// TwinCAT 3 PLC project PLC
// ProgramVersion: 3.1.4026.21
// libraries:
//   Tc2_MC2, * (Beckhoff Automation GmbH)
//   Tc2_Standard, * (Beckhoff Automation GmbH)
//   Tc2_System, * (Beckhoff Automation GmbH)
//   Tc3_IotBase, * (Beckhoff Automation GmbH)
// project tree:
//   DUTs/ E_State.TcDUT
//   GVLs/ IFC_HW.TcGVL
//   / PlcTask.TcTTO
//   POUs/ FB_Abfuellmodul.TcPOU, FB_CNV.TcPOU, FB_Dispenser.TcPOU, FB_IOT.TcPOU, FB_Man_X.TcPOU, FB_RCrtl.TcPOU, FB_StatusLight.TcPOU, FB_TimeOutError.TcPOU, FB_Transport.TcPOU, FB_Vereinzelung.TcPOU, MAIN.TcPOU
// (motion and I/O tree: see PLC project tempmodel)
// real-time tasks:
//   TASK PlcTask: cycle T#10ms, priority 21, ADS port 350
//   TASK PlcTask1: cycle T#10ms, priority 22, ADS port 351
//   TASK PlcTask2: cycle T#10ms, priority 20, ADS port 352
// variable links:
//   LF_System_PLC/LF_System_PLC Instance <-> PLC/PLC Instance
//     PlcTask Inputs/MAIN.bIN_Gripper <-> PlcTask Outputs/IFC_HW.bGripperClosed
//     PlcTask Inputs/MAIN.bIN_Stopper1 <-> PlcTask Outputs/IFC_HW.bBandHub1
//     PlcTask Inputs/MAIN.bIN_Stopper2 <-> PlcTask Outputs/IFC_HW.bBandHub2
//     PlcTask Inputs/MAIN.bIN_Stopper3 <-> PlcTask Outputs/IFC_HW.bBandHub3
//     PlcTask Inputs/MAIN.bIn_LedGreen <-> PlcTask Outputs/IFC_HW.bAmpelGrun
//     PlcTask Inputs/MAIN.bIn_LedRot <-> PlcTask Outputs/IFC_HW.bAmpelRot
//     PlcTask Inputs/MAIN.bIn_LedYellow <-> PlcTask Outputs/IFC_HW.bAmpelGelb
//     PlcTask Inputs/MAIN.bIn_Schleuse1_L1 <-> PlcTask Outputs/IFC_HW.bR1AKT1
//     PlcTask Inputs/MAIN.bIn_Schleuse1_L2 <-> PlcTask Outputs/IFC_HW.bR2AKT1
//     PlcTask Inputs/MAIN.bIn_Schleuse2_L1 <-> PlcTask Outputs/IFC_HW.bR1AKT2
//     PlcTask Inputs/MAIN.bIn_Schleuse2_L2 <-> PlcTask Outputs/IFC_HW.bR2AKT2
//     PlcTask Outputs/MAIN.bEnable <-> PlcTask Inputs/IFC_HW.bEnable
//     PlcTask Outputs/MAIN.bExecute <-> PlcTask Inputs/IFC_HW.bExecute
//     PlcTask Outputs/MAIN.bOUT_CnvNS{1..4} <-> PlcTask Inputs/IFC_HW.bBandSens{1..4}  (4 links)
//     PlcTask Outputs/MAIN.bOUT_SensMaxX <-> PlcTask Inputs/IFC_HW.bManEndXmax
//     PlcTask Outputs/MAIN.bOUT_SensMinX <-> PlcTask Inputs/IFC_HW.bManEndXmin
//     PlcTask Outputs/MAIN.bOut_VereinzelungNS1 <-> PlcTask Inputs/IFC_HW.bEinzelSens1
//     PlcTask Outputs/MAIN.bOut_VereinzelungNS2 <-> PlcTask Inputs/IFC_HW.bEinzelSens2
//     PlcTask Outputs/MAIN.bOut_VereinzelungNS3 <-> PlcTask Inputs/IFC_HW.bEinzelSens3
//     PlcTask Outputs/MAIN.iOut_USS1 <-> PlcTask Inputs/IFC_HW.iFillSens1
//     PlcTask Outputs/MAIN.iOut_USS2 <-> PlcTask Inputs/IFC_HW.iFillSens2
//     PlcTask Outputs/MAIN.iOut_USS3 <-> PlcTask Inputs/IFC_HW.iFillSens3
//   PLC/PLC Instance <-> NC-Task 1 SAF/Axes/BandAchse
//     PlcTask Inputs/IFC_HW.ax_BandMotor.NcToPlc <-> Outputs/ToPlc
//     PlcTask Outputs/IFC_HW.ax_BandMotor.PlcToNc <-> Inputs/FromPlc
//   PLC/PLC Instance <-> NC-Task 1 SAF/Axes/Extruder1
//     PlcTask Inputs/IFC_HW.ax_Extruder1.NcToPlc <-> Outputs/ToPlc
//     PlcTask Outputs/IFC_HW.ax_Extruder1.PlcToNc <-> Inputs/FromPlc
//   PLC/PLC Instance <-> NC-Task 1 SAF/Axes/Extruder2
//     PlcTask Inputs/IFC_HW.ax_Extruder2.NcToPlc <-> Outputs/ToPlc
//     PlcTask Outputs/IFC_HW.ax_Extruder2.PlcToNc <-> Inputs/FromPlc
//   PLC/PLC Instance <-> NC-Task 1 SAF/Axes/Extruder3
//     PlcTask Inputs/IFC_HW.ax_Extruder3.NcToPlc <-> Outputs/ToPlc
//     PlcTask Outputs/IFC_HW.ax_Extruder3.PlcToNc <-> Inputs/FromPlc
//   PLC/PLC Instance <-> NC-Task 1 SAF/Axes/X_Achse_Manipulator
//     PlcTask Inputs/IFC_HW.ax_ManX.NcToPlc <-> Outputs/ToPlc
//     PlcTask Outputs/IFC_HW.ax_ManX.PlcToNc <-> Inputs/FromPlc

CONFIGURATION PLC
    RESOURCE PLC ON TwinCAT3
        TASK PlcTask(INTERVAL := T#10ms, PRIORITY := 20);
        PROGRAM MAIN WITH PlcTask : MAIN;
    END_RESOURCE
END_CONFIGURATION

// ---- DUTs/E_State.TcDUT
{attribute 'qualified_only'}
{attribute 'strict'}
{attribute 'to_string'}
TYPE E_State :
(
    Off,
    Init,
    Ready,
    Production,
    Done,
    Error,
    Stop,
    Setup
);
END_TYPE

// ---- GVLs/IFC_HW.TcGVL
// In dieser GVL werden alle Variablen deklariert die auf die realen Klemmen zugreifen
VAR_GLOBAL
	
	// Allgemeine Variablen fur MAIN und HMI
		bEnable		AT%I*	: BOOL;			// Enable Factory (HMI Production Umgebung)
		bExecute	AT%I*	: BOOL;			// Startsignal	(Start Knopf Konsole)
		bStop				: BOOL;			// Stop Variable (interne Variable um FB's zu stoppen)
		bReset 				: bool; 		// Reset neu hinzugefgt
		
	// Station Statusampel	
		bAmpelRot 	AT%Q* 	: BOOL;			// Signal-LED Rot
		bAmpelGelb 	AT%Q* 	: BOOL;			// Signal-LED Gelb
		bAmpelGrun 	AT%Q* 	: BOOL;			// Signal-LED Grun
			
	// Station Vereinzelung
		bEinzelSens1 	AT%I*	: BOOL;					// Separation Sensor 1 (Kammer)
		bEinzelSens2 	AT%I*	: BOOL;					// Separation Sensor 2 (Rohr)
		bEinzelSens3 	AT%I*	: BOOL;					// Separation Sensor 3 (Flasche auf Kopf)
		bR1AKT1 		AT%Q* 	: BOOL := FALSE;		// Relais 1 Aktor 1 (Schleuse Oben öffnen)
		bR2AKT1 		AT%Q* 	: BOOL := TRUE; 		// Relais 2 Aktor 1 (Schleuse Oben schließen)
		bR1AKT2 		AT%Q* 	: BOOL := FALSE;		// Relais 1 Aktor 2 (Schleuse Unten öffne)
		bR2AKT2 		AT%Q* 	: BOOL := TRUE;			// Relais 2 Aktor 2	(Schleuse Unten schließen)
	
	// Station Forderband
		bBandSens1 	AT %I*	: BOOL;		// Forderband Sensor 1 (Extruder 1)
		bBandSens2	AT %I*	: BOOL;		// Forderband Sensor 2 (Extruder 2)
		bBandSens3 	AT %I*	: BOOL;		// Forderband Sensor 3 (Extruder 3)
		bBandSens4 	AT %I*	: BOOL;		// Forderband Sensor 4 (Übergabe Roboter)
		bBandHub1 	AT %Q*	: BOOL;		// Forderband Hubmagnet 1 (Schleuse Extruder 1)
		bBandHub2 	AT %Q*	: BOOL;		// Forderband Hubmagnet 1 (Schleuse Extruder 2)
		bBandHub3 	AT %Q*	: BOOL;		// Forderband Hubmagnet 1 (Schleuse Extruder 3)
		
		ax_Extruder1 	: AXIS_REF;		// Forderband NC-Achse Extruder 1
		ax_Extruder2 	: AXIS_REF;		// Forderband NC-Achse Extruder 2
		ax_Extruder3 	: AXIS_REF;		// Forderband NC-Achse Extruder 3
		ax_BandMotor 	: AXIS_REF;		// Forderband NC-Achse Band
		
		iBandFullmenge1		: INT := 1;	// in Gramm (Soll Füllmenge Extruder 1)
		iBandFullmenge2		: INT := 1;	// in Gramm (Soll Füllmenge Extruder 2)
		iBandFullmenge3		: INT := 1;	// in Gramm (Soll Füllmenge Extruder 3)
		
	//Füllstandsüberwachung
		iFillSens1 AT%I*	: UINT;		// Füllstandssensor im Granulatspeicher 1
		iFillSens2 AT%I*	: UINT;		// Füllstandssensor im Granulatspeicher 2
		iFillSens3 AT%I*	: UINT;		// Füllstandssensor im Granulatspeicher 3
		
		rFillLevelPercent1	: REAL;		// Füllstand im Granulatspeicher 1 in %
		rFillLevelGramm1	: REAL;		// Füllstand im Granulatspeicher 1 in g
		rFillLevelPercent2	: REAL;		// Füllstand im Granulatspeicher 2 in %
		rFillLevelGramm2	: REAL;		// Füllstand im Granulatspeicher 2 in g
		rFillLevelPercent3	: REAL;		// Füllstand im Granulatspeicher 3 in %
		rFillLevelGramm3	: REAL;		// Füllstand im Granulatspeicher 3 in g
		
		rMaxFillLevel 		: REAL := 375;	// Kalibrierter Füllstand für 10% * 10
		
	// Station Waage
		sWaageNachricht		: STRING;	// Nachricht von Wagezelle (fur virtuelle Inbetriebnahme notig)
		bWaageNull			: BOOL;		// TARA Waage (Waage auf Null setzen)
		iWaageMesswert		: INT;		// Messwert der Waage
		
	// Station Behalteridentifikation
		bIdSensorTrager		: BOOL;		// Sensor bei Erkennung eines Datentrager
		sIdNachricht		: STRING;	// Nachricht von RFID-System (fur virtuelle Inbetriebnahme notig)
		sSeriennummer		: STRING;	// Seriennummer RFID-Tag
		
	//Temperierstation
		bVentilator1 	AT %Q*	: BOOL;		// Ventilator 1
		bVentilator2 	AT %Q*	: BOOL;		// Ventilator 2
		bVentilator3 	AT %Q*	: BOOL;		// Ventilator 3
		
		iTempSens1 		AT%I*	: UINT;		// Temperatursensor 1
		iTempSens2 		AT%I*	: UINT;		// Temperatursensor 2
		iHeizpatrone 	AT%Q*	: UINT;		// Heizpatronen
		
		iMaxTemp				: UINT := 5500;		// in °C * 100
		
	// Station Manipulator
		bManEndXmin 		AT%I* 	: BOOL := TRUE;		// Manipulator min Endschalter Achse x
		bManEndYmin 		AT%I* 	: BOOL := TRUE;		// Manipulator min Endschalter Achse y
		bManEndZmin 		AT%I* 	: BOOL := TRUE;		// Manipulator min Endschalter Achse z
		bManEndGmin 		AT%I* 	: BOOL := TRUE;		// Manipulator min Endschalter Achse Gripper
		bManEndXmax 		AT%I* 	: BOOL := TRUE;		// Manipulator max Endschalter Achse x
		bManEndYmax 		AT%I* 	: BOOL := TRUE;		// Manipulator max Endschalter Achse y
		bManEndZmax 		AT%I* 	: BOOL := TRUE;		// Manipulator max Endschalter Achse z
		bManEndGmax 		AT%I* 	: BOOL := TRUE;		// Manipulator max Endschalter Achse Gripper
		bManBrakeZ			AT%Q*	: BOOL := FALSE;	// Bremse Achse z
		
		ax_ManX			: AXIS_REF;			// Manipulator NC-Achse x
		ax_ManY			: AXIS_REF;			// Manipulator NC-Achse y
		ax_ManZ			: AXIS_REF;			// Manipulator NC-Achse z
		ax_ManG			: AXIS_REF; 		// Manipulator NC-Achse Gripper
		
		bGripperClosed		AT%Q*	: BOOL; 			// signal if gripper is closed ONLY USED IN SIM
END_VAR

// ---- POUs/MAIN.TcPOU
PROGRAM MAIN
VAR
	// Die Logik-Bausteine (Module Level)
    fbAmpel        : FB_StatusLight;
    //fbVereinzelung : FB_Vereinzelung;
    //fbTransport    : FB_Transport;
    
    // NEU: Die drei Abfüllstationen (Dispenser)
    //fbDisp1        : FB_Dispenser;
    //fbDisp2        : FB_Dispenser;
    //fbDisp3        : FB_Dispenser;

    // NEU: Der Werksleiter / Master (Machine Level)
    // Er steuert die oben genannten Module
    fbModul        : FB_Abfuellmodul;
	fbManX         : FB_Man_X;
    // Die Hardware-Übersetzer für die Relais (Process Level)
//     fbRelaisZyl1   : FB_RCrtl; // Schleuse oben
//     fbRelaisZyl2   : FB_RCrtl; // Schleuse unten
    
    // Der Antrieb
    //fbBand         : FB_CNV;
	fbiot : FB_IOT;
	
	//reset
	reset : BOOL;
	bError : Bool;
END_VAR

// --- 1. DER CHEF GIBT DIE BEFEHLE (Hierarchisches Modul) ---

fbiot(iUSS1 := IFC_HW.iFillSens1, iUSS2 := IFC_HW.iFillSens2, iUSS3 := IFC_HW.iFillSens3);
//fbiot(iUSS1 := iIn_USS1, iUSS2 := iIn_USS2, iUSS3 := iIn_USS3);


fbModul(
    bEnable := IFC_HW.bEnable,
    bExecute := IFC_HW.bExecute,
	//bTransportError := fbTransport.bError, 
    bReset := reset,
    
    // Status-Rückmeldungen der Arbeiter abfragen
    //bVereinzelungDone := (fbVereinzelung.eStateOut = E_State.Done),
    //bTransportDone    := (fbTransport.eState = E_State.Done),
    //bDisp1Done        := (fbDisp1.eState = E_State.Done),
    //bDisp2Done        := (fbDisp2.eState = E_State.Done),
    //bDisp3Done        := (fbDisp3.eState = E_State.Done)
);


fbManX(
    // Steuerbefehle
    bEnable         := ifc_hw.bEnable,
    bExecute        := ifc_hw.bExecute, // Hier ggf. eine andere Variable nehmen, wenn er unabhängig vom Abfüllmodul starten soll!
    bHalt           := FALSE,           // Aktuell nicht extern genutzt, ggf. anpassen
    
    // Hardware-Sensoren (Endschalter)
    bEndSchalterMin := ifc_hw.bManEndXmin, 
    bEndSchalterMax := ifc_hw.bManEndXmax, // Falls vorhanden, sonst FALSE
    
    // Fahrparameter (Können später auch aus einer Rezeptur/HMI kommen)
    fPosition       := -500.0,  // Zielposition (Beispiel)
    fVelocity       := 30.0,  // Zielgeschwindigkeit
    pHome           := 0.0,   // Referenzposition am linken Anschlag
    
    // Verknüpfung zur NC-Achse
    ax              := ifc_hw.ax_ManX
);

// --- 2. DIE ARBEITER FÜHREN AUS ---

// Vereinzelung
// fbVereinzelung(
//     bEnable  := IFC_HW.bEnable,
//     bExecute := fbModul.bStartVereinzelung,
//     bSens1   := IFC_HW.bEinzelSens1,
//     bSens2   := IFC_HW.bEinzelSens2,
//     bSens3   := IFC_HW.bEinzelSens3
// );

// Ampel und Relais für Vereinzelung
fbAmpel(eState := fbModul.eState);
IFC_HW.bAmpelRot   := fbAmpel.bLightRed;
IFC_HW.bAmpelGelb  := fbAmpel.bLightYellow;
IFC_HW.bAmpelGrun  := fbAmpel.bLightGreen;

// fbRelaisZyl1(bIn := fbModul.fbVereinzelung.bGate1);
// fbRelaisZyl2(bIn := fbModul.fbVereinzelung.bGate2);
// IFC_HW.bR1AKT1 := fbRelaisZyl1.bQ1;
// IFC_HW.bR2AKT1 := fbRelaisZyl1.bQ2;
// IFC_HW.bR1AKT2 := fbRelaisZyl2.bQ1;
// IFC_HW.bR2AKT2 := fbRelaisZyl2.bQ2;

// Transport-Management
// fbTransport(
//     bEnable  := IFC_HW.bEnable,
//     bExecute := fbModul.bStartTransport,    // <-- Befehl kommt vom Chef
// 	bReset   := reset,
//     nStation := fbModul.nZielStation,       // <-- Ziel (1, 2, 3, 4) kommt vom Chef
//     bSens1   := IFC_HW.bBandSens1,
//     bSens2   := IFC_HW.bBandSens2,
//     bSens3   := IFC_HW.bBandSens3,
//     bSens4   := IFC_HW.bBandSens4
// );

// Die Band-Stopper
// IFC_HW.bBandHub1 := fbTransport.bHub1;
// IFC_HW.bBandHub2 := fbTransport.bHub2;
// IFC_HW.bBandHub3 := fbTransport.bHub3;


// --- 3. DIE EXTRUDER ---

// fbDisp1(
//     ax := IFC_HW.ax_Extruder1,
//     bEnable := IFC_HW.bEnable,
//     bExecute := fbModul.bStartDisp1,        // <-- Befehl kommt vom Chef
//     bSensFlasche := IFC_HW.bBandSens1,
//     iFuellstand := IFC_HW.iFillSens1,
//     iLimit := 80                            // Hier könntest du später Variablen einsetzen
// );
// 
// fbDisp2(
//     ax := IFC_HW.ax_Extruder2,
//     bEnable := IFC_HW.bEnable,
//     bExecute := fbModul.bStartDisp2,        // <-- Befehl kommt vom Chef
//     bSensFlasche := IFC_HW.bBandSens2,
//     iFuellstand := IFC_HW.iFillSens2,
//     iLimit := 80
// );
// 
// fbDisp3(
//     ax := IFC_HW.ax_Extruder3,
//     bEnable := IFC_HW.bEnable,
//     bExecute := fbModul.bStartDisp3,        // <-- Befehl kommt vom Chef
//     bSensFlasche := IFC_HW.bBandSens3,
//     iFuellstand := IFC_HW.iFillSens3,
//     iLimit := 80
// );


// --- 4. DER MUSKEL FÜRS BAND ---

// fbBand(
//     bEnable  := IFC_HW.bEnable,        
//     bExecute := fbModul.fbTransport.bBandExecute, // Fahrbefehl vom Transport-Baustein
//     bHalt    := fbModul.fbTransport.bBandHalt,    // Bremsbefehl vom Transport-Baustein
//     rVel     := 50.0,                 
//     ax       := IFC_HW.ax_BandMotor    
// );

bError := (fbModul.eState = E_State.Error); 	// Überprüfen ob Fehler
ifc_hw.breset := reset;
IF reset AND NOT bError THEN 
	ifc_hw.bStop := FALSE;
	reset := FALSE;
END_IF

END_PROGRAM

// ---- POUs/FB_StatusLight.TcPOU
FUNCTION_BLOCK FB_StatusLight
VAR_INPUT
    eState : E_State;
END_VAR
VAR_OUTPUT
	bLightRed    : BOOL;
    bLightYellow : BOOL;
    bLightGreen  : BOOL;
END_VAR
VAR
	fbTimer      : TON;   // Timer
    bBlinkSignal : BOOL;  // Wechsel
END_VAR

// Grundstellung -> alles aus
bLightRed    := FALSE;
bLightYellow := FALSE;
bLightGreen  := FALSE;

// Blink Signal
fbTimer(IN := NOT fbTimer.Q, PT := T#500MS);
IF fbTimer.Q THEN
    bBlinkSignal := NOT bBlinkSignal;
END_IF

// Blink Zustände
CASE eState OF
    E_State.Off:
        bLightRed := TRUE;
        
    E_State.Production:
        bLightGreen := TRUE;
        
    E_State.Done:
        bLightYellow := TRUE;
        bLightGreen  := TRUE;
	
	E_State.Error:
        bLightRed := bBlinkSignal; // Rot blinken
        
    E_State.Stop:
        bLightRed    := bBlinkSignal; // Rot und Gelb blinken
        bLightYellow := bBlinkSignal;
        
    E_State.Init:
        bLightGreen := bBlinkSignal; // Grün blinken
        
    E_State.Ready:
        bLightYellow := bBlinkSignal; // Gelb und Grün blinken
        bLightGreen  := bBlinkSignal;
        
    E_State.Setup:
        bLightYellow := bBlinkSignal; // Gelb blinken
END_CASE

END_FUNCTION_BLOCK

// ---- POUs/FB_Abfuellmodul.TcPOU
FUNCTION_BLOCK FB_Abfuellmodul
VAR_INPUT
    bEnable  : BOOL;
    bExecute : BOOL;
    bReset   : BOOL;
    
    // Status-Rückmeldungen der Abteilungsleiter
    // bVereinzelungDone : BOOL;
    // bTransportDone    : BOOL;
    // bDisp1Done        : BOOL;
    // bDisp2Done        : BOOL;
    // bDisp3Done        : BOOL;
    
    // Error handling
    //bTransportError : BOOL; 
END_VAR
VAR_OUTPUT
    eState   : E_State;
END_VAR
VAR
    nState : INT;
    i      : INT; // Unser Stations-Zähler (1, 2, 3)
    bFlascheAktiv : BOOL;    // Flasche im System?
    
    fbVereinzelung : FB_Vereinzelung; 
    fbTransport    : FB_Transport;
    fbDisp1        : FB_Dispenser;
    fbDisp2        : FB_Dispenser;
    fbDisp3        : FB_Dispenser;
    
    // Start-Befehle
    bStartVereinzelung : BOOL;
    bStartTransport    : BOOL;
    nZielStation       : INT;     // Welcher Extruder ist das Ziel?
    bStartDisp1        : BOOL;
    bStartDisp2        : BOOL;
    bStartDisp3        : BOOL;
    
    bStop : Bool;
    nMemState: INT;
END_VAR



IF NOT bEnable THEN
    nState := 0;
    eState := E_State.Off;
ELSIF fbTransport.bError AND nState <> 99 THEN
    nMemState := nState;
    nState := 99;
END_IF

// neu 
IF bStop THEN
    nMemState := nState;
END_IF

CASE nState OF
    0: // Start / Bereit
        IF bEnable THEN
            eState := E_State.Ready;
        END_IF
        
        bStartVereinzelung := FALSE;
        bStartTransport    := FALSE;
        bStartDisp1        := FALSE;
        bStartDisp2        := FALSE;
        bStartDisp3        := FALSE;

        IF bExecute THEN
            nState := 10;
        END_IF

    10: // "Vereinzeln der Flasche"
        eState := E_State.Production;
        // --- 1. INTELLIGENTE SUCHE: Steht die Flasche exakt am Sensor? ---
        IF IFC_HW.bBandSens1 THEN
            i := 1; nState := 30; 
        ELSIF IFC_HW.bBandSens2 THEN
            i := 2; nState := 30; 
        ELSIF IFC_HW.bBandSens3 THEN
            i := 3; nState := 30; 
        ELSIF IFC_HW.bBandSens4 THEN
            nState := 40; 

        // --- 2. Suche im Gedächtnis (Der Blinde Fleck) ---
        ELSIF bFlascheAktiv THEN
            // Sensoren sehen nichts, aber da ist eine Flasche!
            // WICHTIG: Wohin war sie gerade unterwegs?
            IF i < 4 THEN
                nState := 20; // Sie war auf dem Weg zu einem Extruder (1, 2 oder 3)
            ELSE
                nState := 40; // Sie war schon auf der Zielgeraden zum Roboter (Station 4)
            END_IF
            
        // --- 3. NORMALBETRIEB: Keine alte Flasche im System ---
        ELSE
            bStartVereinzelung := TRUE;
        END_IF

        IF fbVereinzelung.eStateOut = E_State.Done THEN
            bFlascheAktiv := TRUE;
            i := 1;                      // Zähler auf ersten Extruder setzen!
            nState := 20;
        END_IF

    20: // "Fördern zu Extruder i"
        eState := E_State.Production;
        nZielStation := i; // Dem Transport das Ziel (1, 2 oder 3) mitteilen
        bStartTransport := TRUE;

        IF fbTransport.eState = E_State.Done THEN
            
               IF i = 1 THEN
                bStartVereinzelung := FALSE; // Vereinzelung darf nächste Flasche holen
            END_IF
            
            bStartTransport := FALSE;
            nState := 30;
        END_IF

    30: // "Extruder i Start"
        eState := E_State.Production;
        // Welcher Dispenser muss gestartet werden?
        IF i = 1 THEN bStartDisp1 := TRUE; END_IF
        IF i = 2 THEN bStartDisp2 := TRUE; END_IF
        IF i = 3 THEN bStartDisp3 := TRUE; END_IF

        // Warten, bis der jeweilige Extruder "fertig" meldet
        IF (i = 1 AND fbDisp1.eState = E_State.Done) OR
           (i = 2 AND fbDisp2.eState = E_State.Done) OR
           (i = 3 AND fbDisp3.eState = E_State.Done) THEN
            
            // Befehle wieder wegnehmen
            bStartDisp1 := FALSE;
            bStartDisp2 := FALSE;
            bStartDisp3 := FALSE;

            // Zähler erhöhen! (i = i + 1)
            i := i + 1;

            // Prüfen, ob wir alle 3 Extruder durch haben
            IF i < 4 THEN
                nState := 20; // Zurück zu Schritt 20: Fördern zum NÄCHSTEN Extruder!
            ELSE
                nState := 40; // Alle 3 Farben sind drin! Weiter zur Übergabe.
            END_IF
        END_IF

    40: // "Übergabe zu Portalroboter" / Station 4
        eState := E_State.Production;
        nZielStation := 4;
        bStartTransport := TRUE;

        IF fbTransport.eState = E_State.Done THEN
            bStartTransport := FALSE;
            nState := 50;
        END_IF

    50: // Done
        eState := E_State.Done;
        bFlascheAktiv := FALSE; 

        IF NOT bExecute THEN
            nState := 0; 
        END_IF
    
    99: // Error
        eState := E_State.Error; 
        IF NOT fbTransport.bError THEN
            nState := nMemState; // Nach Reset zurück zum alten zustand
        END_IF
        
END_CASE

// FBs

fbVereinzelung(
    bEnable  := bEnable,
    bExecute := bStartVereinzelung, // Interne Variable
    bSens1   := IFC_HW.bEinzelSens1,
    bSens2   := IFC_HW.bEinzelSens2,
    bSens3   := IFC_HW.bEinzelSens3
);

fbTransport(
    bEnable  := bEnable,
    bExecute := bStartTransport,    // Interne Variable
    bReset   := bReset,
    nStation := nZielStation,       // Interne Variable
    bSens1   := IFC_HW.bBandSens1,
    bSens2   := IFC_HW.bBandSens2,
    bSens3   := IFC_HW.bBandSens3,
    bSens4   := IFC_HW.bBandSens4
);

// Direktes Beschreiben der Hardware-Ausgänge für den Transport
IFC_HW.bBandHub1 := fbTransport.bHub1;
IFC_HW.bBandHub2 := fbTransport.bHub2;
IFC_HW.bBandHub3 := fbTransport.bHub3;

fbDisp1(
    ax := IFC_HW.ax_Extruder1,
    bEnable := bEnable,
    bExecute := bStartDisp1,        // Interne Variable
    bSensFlasche := IFC_HW.bBandSens1,
    iFuellstand := IFC_HW.iFillSens1,
    iLimit := 80
);

fbDisp2(
    ax := IFC_HW.ax_Extruder2,
    bEnable := bEnable,
    bExecute := bStartDisp2,        // Interne Variable
    bSensFlasche := IFC_HW.bBandSens2,
    iFuellstand := IFC_HW.iFillSens2,
    iLimit := 80
);

fbDisp3(
    ax := IFC_HW.ax_Extruder3,
    bEnable := bEnable,
    bExecute := bStartDisp3,        // Interne Variable
    bSensFlasche := IFC_HW.bBandSens3,
    iFuellstand := IFC_HW.iFillSens3,
    iLimit := 80
);

END_FUNCTION_BLOCK

// ---- POUs/FB_Vereinzelung.TcPOU
FUNCTION_BLOCK FB_Vereinzelung
VAR_INPUT
	bEnable  : BOOL; // Anlage aktiv
    bExecute : BOOL; // Startschalter
    bSens1   : BOOL; // Flasche in Kammer
    bSens2   : BOOL; // Flasche im Speicher
    bSens3   : BOOL; // Flasche am Band
END_VAR
VAR_OUTPUT
	
    eStateOut : E_State; // Aktueller Betriebszustand
END_VAR
VAR
	nState  : INT := 0;  // Speichert unseren aktuellen Schritt (0, 10, 11, ...)
    fbTimer : TON;       // Timer für die Wartezeiten der Zylinder
	bGate1    : BOOL;    // Befehl: Schleuse 1 öffnen
    bGate2    : BOOL;    // Befehl: Schleuse 2 öffnen
	fbRelaisZyl1   : FB_RCrtl; // Schleuse oben
    fbRelaisZyl2   : FB_RCrtl; // Schleuse unten
	
END_VAR

// Timer Starten
fbTimer();

// Instanzierung Schläusen
fbRelaisZyl1(bIn := bGate1);
fbRelaisZyl2(bIn := bGate2);
IFC_HW.bR1AKT1 := fbRelaisZyl1.bQ1;
IFC_HW.bR2AKT1 := fbRelaisZyl1.bQ2;
IFC_HW.bR1AKT2 := fbRelaisZyl2.bQ1;
IFC_HW.bR2AKT2 := fbRelaisZyl2.bQ2;

// Not-Aus
IF NOT bEnable THEN
    nState := 0;
END_IF

// State Machine
CASE nState OF
    0: // Off
        bGate1 := FALSE;
        bGate2 := FALSE;
        eStateOut := E_State.Off;
        
        IF bEnable AND bSens2 THEN
            nState := 10;
        END_IF
        
     9: // Gates schließen
        bGate1 := FALSE;
        bGate2 := FALSE;
        
        fbTimer(IN := TRUE, PT := T#1S); 
        
        IF fbTimer.Q THEN
            nState := 10;
            fbTimer(IN := FALSE);
        END_IF
        
    10: // Schleuse 1 auf, warten auf Flasche
        bGate1 := TRUE;
        bGate2 := FALSE;
        eStateOut := E_State.Init;
        
        IF bSens3 THEN
            nState := 11;
            fbTimer(IN := FALSE);
        END_IF
        
    11: // Schleuse 1 schließen
        bGate1 := FALSE;
        bGate2 := FALSE;
        eStateOut := E_State.Init;
        fbTimer(IN := TRUE, PT := T#1S); // 1 Sekunde warten, bis Zylinder mechanisch zu ist
        
        IF fbTimer.Q THEN
            nState := 20;
            fbTimer(IN := FALSE);
        END_IF
        
    20: // Warten auf bExecute
        bGate1 := FALSE;
        bGate2 := FALSE;
        eStateOut := E_State.Ready; // Ampel Gelb/Grün
        
        IF bExecute THEN
            nState := 30;
            fbTimer(IN := FALSE);
        END_IF
        
    30: // Schleuse 2 öffnen
        bGate1 := FALSE;
        bGate2 := TRUE;
        eStateOut := E_State.Production; 
       	
        fbTimer(IN := TRUE, PT := T#0.5S);	//Timer für Fallzeit
        
        IF fbTimer.Q THEN
            nState := 40;
            fbTimer(IN := FALSE);
        END_IF
        
    40: // Done zurückgeben.
        bGate1 := FALSE;
        eStateOut := E_State.Done;
        
        IF NOT bExecute THEN
            nState := 9; 
        END_IF
        
END_CASE

END_FUNCTION_BLOCK

// ---- POUs/FB_RCrtl.TcPOU
FUNCTION_BLOCK FB_RCrtl
VAR_INPUT
	bIn : BOOL; // TRUE = Öffnen, FALSE = Schließen
END_VAR
VAR_OUTPUT
	bQ1 : BOOL; // Relais 1
    bQ2 : BOOL; // Relais 2
END_VAR
VAR
END_VAR

IF bIn THEN
    bQ1 := TRUE;
    bQ2 := FALSE;
ELSIF NOT bIn THEN
    bQ1 := FALSE;
    bQ2 := TRUE;
END_IF

END_FUNCTION_BLOCK

// ---- POUs/FB_Transport.TcPOU
FUNCTION_BLOCK FB_Transport
VAR_INPUT
    bEnable   : BOOL;
    bExecute  : BOOL;
	bReset : BOOL; // um Fehler zurück zusetzen
    nStation  : INT; // ZielStation
    
    // Lichtschranken
    bSens1    : BOOL;
    bSens2    : BOOL;
    bSens3    : BOOL;
    bSens4    : BOOL;
END_VAR
VAR_OUTPUT
    eState    : E_State;
    
    // Hubs
    bHub1     : BOOL;
    bHub2     : BOOL;
    bHub3     : BOOL;
	
	
	bError: BOOL;
	ErrorID: DWORD;
END_VAR
VAR
    nState : INT;
	nMemState: INT;
	fbTO_Transport : FB_TimeOutError(9001,T#10S); // Error wenn zu Flasche zulange braucht
	
	bBandExecute : BOOL;
	bBandHalt    : BOOL;
    
	bStop : BOOL;
	fbBand : FB_CNV;
END_VAR

fbTO_Transport(
	bIN:= eState = E_State.Production, 
	bZiel:= eState = E_State.Done, 
	bReset:= bReset , 
	bError=> bError, 
	ErrorID=> ErrorID);

fbBand(
    bEnable  := IFC_HW.bEnable,        
    bExecute := bBandExecute, // Fahrbefehl vom Transport-Baustein
    bHalt    := bBandHalt,    // Bremsbefehl vom Transport-Baustein
    rVel     := 50.0,                 
    ax       := IFC_HW.ax_BandMotor    
);

// Übergeordnete Sicherheit
IF NOT bEnable THEN
    nState := 0;
ELSIF bError AND nState <> 99 AND nState <> 100 THEN
	nMemState := nState;
    nState := 99; //Timeout
END_IF

bStop := ifc_Hw.bStop;

CASE nState OF
    0: // Ready
        eState := E_State.Ready;
        bBandExecute := FALSE;
        bBandHalt := FALSE;
        
        // Zylinder geschlossen
        bHub1 := FALSE;
        bHub2 := FALSE;
        bHub3 := FALSE;

        IF bExecute AND nStation > 0 THEN
            nState := 1;
        END_IF

    1: // Öffnen Hubzylinder  
        eState := E_State.Production;
       
        IF nStation = 2 THEN bHub1 := TRUE; END_IF
        IF nStation = 3 THEN bHub2 := TRUE; END_IF
        IF nStation = 4 THEN bHub3 := TRUE; END_IF
        
        nState := 2;
        
    2: // Start Conveyor 
		eState := E_State.Production;
       	bBandExecute := TRUE;
        nState := 3;
        
    3: // Production
		eState := E_State.Production;
        IF (nStation = 1 AND bSens1) OR
           (nStation = 2 AND bSens2) OR
           (nStation = 3 AND bSens3) OR
           (nStation = 4 AND bSens4) THEN
            nState := 4;
        END_IF

    4: // Schließen Hubzylinder
        bHub1 := FALSE;
        bHub2 := FALSE;
        bHub3 := FALSE;
        nState := 5;

    5: // Stop Conveyor 
		bBandExecute := FALSE;
		bBandHalt := TRUE; // Bremsbefehl
        nState := 6;
        
    6: // Done
        eState := E_State.Done;
        bBandHalt := FALSE;
        
        IF NOT bExecute THEN
            nState := 0;
        END_IF
	99: // Error State 
        eState := E_State.Error;
        bBandExecute := FALSE; 
        bBandHalt    := TRUE; 
        
        // Schleusen schließen
        bHub1 := FALSE;
        bHub2 := FALSE;
        bHub3 := FALSE;

        IF bReset THEN 
            nState := 100;
        END_IF

    100: // Reset
        bBandHalt := FALSE;
        IF NOT bError THEN 
            IF nMemState = 3 THEN
                nState := 2;
            ELSE
                nState := nMemState;   
            END_IF 
        END_IF
END_CASE

END_FUNCTION_BLOCK

// ---- POUs/FB_TimeOutError.TcPOU
FUNCTION_BLOCK FB_TimeOutError
VAR_INPUT
	bIN : BOOL;
	bZiel : BOOL;
	bReset : BOOL;
END_VAR
VAR_OUTPUT
	bError : BOOL;
	ErrorID : DWORD;
END_VAR
VAR
	timer : TON;
	_ErrorID : DWORD;
	_PT : TIME;
END_VAR

timer(IN:= , PT:=_PT , Q=> , ET=> );

IF bIN THEN
	timer.IN := TRUE;
END_IF

IF bZiel THEN
	timer.IN := FALSE;
END_IF

IF timer.Q THEN
	bError := TRUE;
	ErrorID := _ErrorID;
	timer.IN := FALSE;
ELSIF bReset THEN
	bError := FALSE;
	ErrorID := 0;
END_IF

//FB_Init is always available implicitly and it is used primarily for initialization.
//The return value is not evaluated. For a specific influence, you can also declare the
//methods explicitly and provide additional code there with the standard initialization
//code. You can evaluate the return value.
METHOD FB_Init: BOOL
VAR_INPUT
    bInitRetains: BOOL; // TRUE: the retain variables are initialized (reset warm / reset cold)
    bInCopyCode: BOOL;  // TRUE: the instance will be copied to the copy code afterward (online change)   
	ErrorID : DWORD;
	PT : time;
END_VAR
_ErrorID := ErrorID;
_PT := PT;
END_METHOD

END_FUNCTION_BLOCK

// ---- POUs/FB_CNV.TcPOU
FUNCTION_BLOCK FB_CNV
VAR_INPUT
	// Steuereingänge
	bEnable : BOOL;
	bExecute : BOOL;
	bHalt : BOOL;
	//Bewegungseigenschaften
	rVel : REAL;
END_VAR
VAR_OUTPUT
	eState : E_State;
END_VAR
VAR
	nState : INT;
	mcPower : MC_Power;
	mcReset : MC_Reset;
	mcVelocity : MC_MoveVelocity;
	mcHalt : MC_Halt;
	mcStop : MC_Stop;
	bStop : BOOL;
END_VAR
VAR_IN_OUT
	ax : Axis_Ref;
END_VAR

// Fehlerüberwachung
IF ax.Status.Error AND nState <> 100 THEN
    nState := 99;
END_IF

bStop := ifc_Hw.bStop;

// States
CASE nState OF
    0: // Off
        eState := E_State.Off;
        mcPower.Enable := FALSE;
        mcPower.Enable_Positive := FALSE;
        mcPower.Enable_Negative := FALSE;
        mcVelocity.Execute := FALSE;
        mcHalt.Execute := FALSE;
        mcReset.Execute := FALSE;
        
        IF bEnable THEN
            nState := 1;
        END_IF
		
		
        
    1: // Init 
        eState := E_State.Init;
        mcPower.Enable := TRUE;
        mcPower.Enable_Positive := TRUE;
        mcPower.Enable_Negative := TRUE;
        
        IF mcPower.Status THEN // State übergang
            nState := 2;
        END_IF
        
        // abbruch
        IF NOT bEnable THEN nState := 0; END_IF 
        
    2: // Ready 
        eState := E_State.Ready;
        mcVelocity.Execute := FALSE;
        mcHalt.Execute := FALSE;
        
        IF bExecute THEN
            nState := 3; // State übergang
        END_IF
        
        // abbruch
        IF NOT bEnable THEN nState := 0; END_IF 
        
    3: // CNV an 
        eState := E_State.Production;
        mcVelocity.Velocity := rVel;
        mcVelocity.Direction := MC_Positive_Direction;
        mcVelocity.Execute := TRUE;
        
        // abbruch mit abbremsen
        IF bHalt OR NOT bEnable THEN
            nState := 4;
        END_IF
        
    4: // CNV aus 
        eState := E_State.Production;
        mcVelocity.Execute := FALSE;
        mcHalt.Execute := TRUE; // Bremsvorgang einleiten
        
        IF mcHalt.Done THEN 
            nState := 5;
        END_IF
        
    5: // Done 
        eState := E_State.Done;
        mcHalt.Execute := FALSE;
        
        IF NOT bEnable THEN
            nState := 0; 
        ELSIF NOT bExecute AND NOT bHalt THEN
            nState := 2; // Wieder zurück auf Ready
        END_IF
		
	80: // Stop CNV
		mcVelocity.Execute := FALSE;
		mcHalt.Execute := FALSE;
		mcStop.Execute := TRUE;
		
		IF mcStop.Done AND NOT bStop THEN
			nState := 81;
		END_IF
        
	81: 
		mcVelocity.Execute := FALSE;
		mcHalt.Execute := FALSE;
		mcStop.Execute := TRUE;
		mcReset.Execute := TRUE;
		
		IF mcReset.Done THEN
			nState := 3;
		END_IF
	
    99: // Error State
        eState := E_State.Error;
        mcPower.Enable := FALSE;
        mcPower.Enable_Positive := FALSE;
        mcPower.Enable_Negative := FALSE;
        mcVelocity.Execute := FALSE;
        mcHalt.Execute := FALSE;
        
        IF bEnable THEN 
            nState := 100;
        END_IF
        
    100: // Resolve 
        mcReset.Execute := TRUE;
        
        IF mcReset.Done THEN
            mcReset.Execute := FALSE;
            nState := 1; // Neustart nach Reset
        ELSIF mcReset.Error THEN
            mcReset.Execute := FALSE;
            nState := 99; // Reset fehlgeschlagen
        END_IF
        
END_CASE

// Bausteine aufrufen
mcPower(Axis := ax, Enable := mcPower.Enable, Enable_Positive := mcPower.Enable_Positive, Enable_Negative := mcPower.Enable_Negative, Override := 100.0);
mcReset(Axis := ax, Execute := mcReset.Execute);
mcVelocity(Axis := ax, Execute := mcVelocity.Execute, Velocity := mcVelocity.Velocity, Direction := mcVelocity.Direction);
mcHalt(Axis := ax, Execute := mcHalt.Execute);

END_FUNCTION_BLOCK

// ---- POUs/FB_Dispenser.TcPOU
FUNCTION_BLOCK FB_Dispenser
VAR_IN_OUT
    ax : AXIS_REF;
END_VAR
VAR_INPUT
    bEnable      : BOOL;
    bExecute     : BOOL;
    bSensFlasche : BOOL; 
    iFuellstand  : UINT; 
    iLimit       : UINT; 
END_VAR
VAR_OUTPUT
    eState       : E_State;
END_VAR
VAR
    nState    : INT;
    mcPower   : MC_Power;          
    mcMove    : MC_MoveRelative;
	mcReset : MC_Reset;
    bMoveExec : BOOL;
END_VAR

// Fehlerabfrage
IF ax.Status.Error AND nState <> 100 THEN
    nState := 99; 
END_IF

// State Machine
CASE nState OF
    0: // Grundstellung
        eState := E_State.Off;
        bMoveExec := FALSE; 
        mcPower.Enable := FALSE;
        
        IF bEnable THEN nState := 1; END_IF

    1: // Warten auf Startsignal
        eState := E_State.Ready;
        mcPower.Enable := TRUE;
        
        IF NOT bEnable THEN nState := 0; END_IF
        IF bExecute THEN nState := 2; END_IF

    2: // Warten auf Flasche
        IF NOT bEnable THEN nState := 0; END_IF
        
        IF bSensFlasche THEN
            nState := 3;
        END_IF

    3: // Befüllen der Flasche
        eState := E_State.Production;
        bMoveExec := TRUE; 
        
        IF mcMove.Done THEN
            bMoveExec := FALSE; 
            nState := 4;
        END_IF
        
        IF mcMove.Error OR ax.Status.Error THEN
            bMoveExec := FALSE; 
            nState := 99; // Error-State
        END_IF

    4: // Fertig
        eState := E_State.Done;
        
        IF NOT bEnable THEN nState := 0; END_IF
        IF NOT bExecute THEN nState := 1; END_IF
        
    99: // Error
        eState := E_State.Error;
        bMoveExec := FALSE;
        mcPower.Enable := FALSE;
        mcReset.Execute := FALSE;
        
		// Reset bei bEnable
        IF bEnable THEN 
            nState := 100; 
        END_IF
        
    100: // Reset
        mcReset.Execute := TRUE;
        
        IF mcReset.Done THEN	// Erfolgreich -> Grundstellung
            mcReset.Execute := FALSE;
            nState := 0;
            
        ELSIF mcReset.Error THEN	// Fehler -> ErrorState
            mcReset.Execute := FALSE;
            nState := 99;
        END_IF
        
END_CASE

mcPower(
    Axis := ax, 
    Enable_Positive := TRUE, 
    Enable_Negative := TRUE, 
    Override := 100.0
);

mcMove(
    Axis := ax, 
    Execute := bMoveExec,
    Distance := 1440.0,      // Umdrehungen
    Velocity := 360.0,      // Umdrehungen pro Sekunde
    Acceleration := 2000.0,
    Deceleration := 2000.0
);

mcReset(
    Axis := ax, 
    Execute := mcReset.Execute
);

END_FUNCTION_BLOCK

// ---- POUs/FB_Man_X.TcPOU
FUNCTION_BLOCK FB_Man_X
VAR_INPUT
    bEnable         : BOOL;  // Reglerfreigabe generelle
    bExecute        : BOOL;  // Startet die absolute Positionierfahrt
    bHalt           : BOOL;  // Sanftes Abbremsen (für normalen Ablauf)
    
    // Sensoren (True = betätigt / belegt)
    bEndSchalterMin : BOOL;  // Linker Endschalter (Gleichzeitig unser Referenzschalter!)
    bEndSchalterMax : BOOL;  // Rechter Endschalter
    bSens4          : BOOL;  // Sensor Bandende
    
    // Fahrparameter
    fPosition       : LREAL; // Zielposition für die absolute Fahrt
    fVelocity       : LREAL; // Zielgeschwindigkeit
    pHome           : LREAL; // Positionswert, der bei Referenzierung gesetzt wird (z.B. 0.0)
END_VAR

VAR_OUTPUT
    eState          : E_State; // Zustandsausgabe für die Main
    fActPos         : LREAL;   // Aktuelle Position für die Anzeige (X)
    
    // Greifer und Freigabe
    bGreifer        : BOOL;    // TRUE = Greifer zu, FALSE = Greifer auf
    bBandFrei       : BOOL;    // TRUE = Flasche weg, nächstes Modul darf starten!
END_VAR

VAR_IN_OUT
    ax              : AXIS_REF; // Verknüpfung zur NC-Achse X
    axY             : AXIS_REF; // Verknüpfung zur virtuellen Achse Y
    axZ             : AXIS_REF; // Verknüpfung zur virtuellen Achse Z
END_VAR

VAR
    // Interne State-Machine Variablen
    nState          : INT;
    bStop           : BOOL;     // Lokale Kopie vom globalen Not-Halt (aus ifc_hw.bStop)
    fbTimer         : TON;      // Timer für das Greifen/Loslassen

    // --- Motion Control Bausteine (X-Achse) ---
    mcPower         : MC_Power;
    mcReset         : MC_Reset;
    mcVelocity      : MC_MoveVelocity; 
    mcMoveAbs       : MC_MoveAbsolute; 
    mcHalt          : MC_Halt;         
    mcStop          : MC_Stop;         
    mcSetPos        : MC_SetPosition;  

    // --- Motion Control Bausteine (Y-Achse virtuell) ---
    mcPowerY        : MC_Power;
    mcMoveAbsY      : MC_MoveAbsolute;

    // --- Motion Control Bausteine (Z-Achse virtuell) ---
    mcPowerZ        : MC_Power;
    mcMoveAbsZ      : MC_MoveAbsolute;
END_VAR



// Timer für den Greifer aufrufen
fbTimer();

// Fehlerüberwachung (Sammelt Errors von ALLEN genutzten Achsen und MC-Bausteinen)
IF (ax.Status.Error OR axY.Status.Error OR axZ.Status.Error OR mcMoveAbs.Error OR mcVelocity.Error OR mcSetPos.Error) AND nState <> 100 THEN
    nState := 99;
END_IF

bStop := ifc_Hw.bStop; // Globale Stop-Variable einlesen

// Stopen über Not-Aus (bStop) oder bEnable weg
IF (bStop OR NOT bEnable) AND nState >= 3 AND nState < 80 THEN
    nState := 80; 
END_IF

// ==========================================
// STATE MACHINE
// ==========================================
CASE nState OF
    0: // Off
        eState := E_State.Off;
        bBandFrei := FALSE;
        bGreifer  := FALSE;
        
        mcPower.Enable := FALSE;
        mcVelocity.Execute := FALSE;
        mcMoveAbs.Execute := FALSE;
        mcHalt.Execute := FALSE;
        mcStop.Execute := FALSE;
        mcReset.Execute := FALSE;
        mcSetPos.Execute := FALSE;
        
        IF bEnable THEN
            nState := 1;
        END_IF
        
    1: // Init (Power On)
        eState := E_State.Init;
        mcPower.Enable := TRUE; // Startet auch Y und Z unten!
        
        IF mcPower.Status THEN 
            nState := 10; // Gehe zur Referenzfahrt für X
        END_IF
        IF NOT bEnable THEN nState := 0; END_IF 
        
    // ==========================================
    // REFERENZFAHRT (Nur X-Achse benötigt das wirklich)
    // ==========================================
    10: // Homing Start (Fahrt nach links)
        eState := E_State.Init; 
        mcVelocity.Velocity := 15.0; 
        mcVelocity.Direction := MC_Negative_Direction; // Nach links zum Min-Schalter
        mcVelocity.Execute := TRUE;
        
        IF NOT bEndSchalterMin THEN
            mcVelocity.Execute := FALSE;
            nState := 11;
        END_IF

    11: // Homing Stop (Am Schalter anhalten)
        mcHalt.Execute := TRUE;
        IF mcHalt.Done THEN
            mcHalt.Execute := FALSE;
            nState := 12;
        END_IF

    12: // Position auf pHome (0.0) nullen
        mcSetPos.Position := pHome;
        mcSetPos.Execute := TRUE;
        
        IF mcSetPos.Done THEN
            mcSetPos.Execute := FALSE;
            nState := 2; // Referenzfahrt fertig -> Ready!
        END_IF
        
    // ==========================================
    // NORMALBETRIEB (Warten auf Flasche)
    // ==========================================
    2: // Ready 
        eState := E_State.Ready;
        mcVelocity.Execute := FALSE;
        mcHalt.Execute := FALSE;
        mcStop.Execute := FALSE;
        bBandFrei := FALSE; // Blockiert das Band, solange wir warten
        
        // Der Manipulator startet jetzt vollautomatisch, sobald die Flasche ankommt!
        IF bSens4 THEN
            nState := 20;
        END_IF
        IF NOT bEnable THEN nState := 0; END_IF
        
    // ==========================================
    // ZYKLUS: PICK & PLACE (Die Choreografie)
    // ==========================================
    20: // 1. Z-Achse nach unten fahren (zur Flasche)
        eState := E_State.Production;
        mcMoveAbsZ.Position := 100.0; // TIEFE ANPASSEN WENN NÖTIG!
        mcMoveAbsZ.Velocity := 150.0;
        mcMoveAbsZ.Execute  := TRUE;
        
        IF mcMoveAbsZ.Done THEN
            mcMoveAbsZ.Execute := FALSE;
            nState := 21;
        END_IF

    21: // 2. Flasche greifen
        bGreifer := TRUE; 
        fbTimer(IN := TRUE, PT := T#0.5S); // Warten bis Greifer mechanisch zu ist
        
        IF fbTimer.Q THEN
            fbTimer(IN := FALSE);
            nState := 22;
        END_IF

    22: // 3. Z-Achse wieder hochfahren
        mcMoveAbsZ.Position := 0.0; // Zurück auf Null (Oben)
        mcMoveAbsZ.Execute  := TRUE;
        
        IF mcMoveAbsZ.Done THEN
            mcMoveAbsZ.Execute := FALSE;
            
            // WICHTIG: Flasche ist in der Luft! Das Band darf weiterarbeiten!
            bBandFrei := TRUE; 
            nState := 23;
        END_IF

    23: // 4. X nach rechts UND Y nach hinten fahren (Gleichzeitig!)
        // X fährt auf Endschalter Max
        mcVelocity.Velocity  := 150.0;
        mcVelocity.Direction := MC_Positive_Direction;
        mcVelocity.Execute   := TRUE;
        
        // Y fährt auf Position
        mcMoveAbsY.Position := 200.0; // Y-TIEFE INS LAGER ANPASSEN!
        mcMoveAbsY.Velocity := 150.0;
        mcMoveAbsY.Execute  := TRUE;
        
        // Warten, bis BEIDE angekommen sind (X am Sensor, Y am Ziel)
        IF NOT bEndSchalterMax AND mcMoveAbsY.Done THEN 
            mcVelocity.Execute := FALSE;
            mcMoveAbsY.Execute := FALSE;
            mcHalt.Execute     := TRUE; // X-Achse abbremsen
            nState := 24;
        END_IF

    24: // 5. Warten bis X-Achse steht
        IF mcHalt.Done THEN
            mcHalt.Execute := FALSE;
            nState := 25;
        END_IF

    25: // 6. Z-Achse nach unten (ins Lager)
        mcMoveAbsZ.Position := 100.0; 
        mcMoveAbsZ.Execute  := TRUE;
        
        IF mcMoveAbsZ.Done THEN
            mcMoveAbsZ.Execute := FALSE;
            nState := 26;
        END_IF

    26: // 7. Flasche loslassen
        bGreifer := FALSE;
        fbTimer(IN := TRUE, PT := T#0.5S); // Warten bis Greifer offen ist
        
        IF fbTimer.Q THEN
            fbTimer(IN := FALSE);
            nState := 27;
        END_IF

    27: // 8. Z-Achse wieder hoch (ohne Flasche)
        mcMoveAbsZ.Position := 0.0; 
        mcMoveAbsZ.Execute  := TRUE;
        
        IF mcMoveAbsZ.Done THEN
            mcMoveAbsZ.Execute := FALSE;
            nState := 28;
        END_IF

    28: // 9. X und Y zurück zur Grundstellung (Gleichzeitig!)
        mcVelocity.Direction := MC_Negative_Direction; // X nach links
        mcVelocity.Execute   := TRUE;
        
        mcMoveAbsY.Position := 0.0; // Y wieder nach vorne
        mcMoveAbsY.Execute  := TRUE;
        
        IF NOT bEndSchalterMin AND mcMoveAbsY.Done THEN 
            mcVelocity.Execute := FALSE;
            mcMoveAbsY.Execute := FALSE;
            mcHalt.Execute     := TRUE;
            nState := 29;
        END_IF

    29: // 10. Warten bis X steht -> Fertig!
        IF mcHalt.Done THEN
            mcHalt.Execute := FALSE;
            bBandFrei := FALSE; // Reset für den nächsten Durchlauf
            nState := 2; // Zurück auf Lauerstellung!
        END_IF
        
    // ==========================================
    // NOT-HALT / STOP
    // ==========================================
    80: // Stop Achse (Harter Stopp)
        mcMoveAbs.Execute := FALSE;
        mcVelocity.Execute := FALSE;
        mcHalt.Execute := FALSE;
        mcMoveAbsY.Execute := FALSE;
        mcMoveAbsZ.Execute := FALSE;
        mcStop.Execute := TRUE;
        
        IF mcStop.Done AND NOT bStop THEN
            nState := 81;
        END_IF
        
    81: // Stop lösen
        mcStop.Execute := FALSE; 
        nState := 1; // Sicherer Neustart inkl. Homing
    
    // ==========================================
    // ERROR HANDLING
    // ==========================================
    99: // Error State
        eState := E_State.Error;
        mcPower.Enable := FALSE;
        mcVelocity.Execute := FALSE;
        mcMoveAbs.Execute := FALSE;
        mcMoveAbsY.Execute := FALSE;
        mcMoveAbsZ.Execute := FALSE;
        mcHalt.Execute := FALSE;
        mcStop.Execute := FALSE;
        
        IF bEnable THEN 
            nState := 100;
        END_IF
        
    100: // Resolve / Reset
        mcReset.Execute := TRUE;
        
        IF mcReset.Done THEN
            mcReset.Execute := FALSE;
            nState := 1; // Neustart
        ELSIF mcReset.Error THEN
            mcReset.Execute := FALSE;
            nState := 99; // Reset fehlgeschlagen
        END_IF
        
END_CASE

// ==========================================
// BAUSTEINE AUFRUFEN (Am Ende des Zyklus)
// ==========================================

// --- X-ACHSE ---
mcPower(
    Axis            := ax, 
    Enable          := mcPower.Enable, 
    Enable_Positive := mcPower.Enable AND bEndSchalterMax, 
    Enable_Negative := mcPower.Enable AND bEndSchalterMin, 
    Override        := 100.0
);
mcReset(Axis := ax, Execute := mcReset.Execute);
mcVelocity(Axis := ax, Execute := mcVelocity.Execute, Velocity := mcVelocity.Velocity, Direction := mcVelocity.Direction);
mcMoveAbs(Axis := ax, Execute := mcMoveAbs.Execute, Position := mcMoveAbs.Position, Velocity := mcMoveAbs.Velocity);
mcHalt(Axis := ax, Execute := mcHalt.Execute);
mcStop(Axis := ax, Execute := mcStop.Execute);
mcSetPos(Axis := ax, Execute := mcSetPos.Execute, Position := mcSetPos.Position);
fActPos := ax.NcToPlc.ActPos;

// --- Y-ACHSE (Virtuell) ---
mcPowerY(
    Axis            := axY, 
    Enable          := mcPower.Enable, 
    Enable_Positive := mcPower.Enable, // Keine Sensoren -> Immer TRUE solange Enable
    Enable_Negative := mcPower.Enable,
    Override        := 100.0
);
mcMoveAbsY(Axis := axY, Execute := mcMoveAbsY.Execute, Position := mcMoveAbsY.Position, Velocity := mcMoveAbsY.Velocity);

// --- Z-ACHSE (Virtuell) ---
mcPowerZ(
    Axis            := axZ, 
    Enable          := mcPower.Enable, 
    Enable_Positive := mcPower.Enable,
    Enable_Negative := mcPower.Enable,
    Override        := 100.0
);
mcMoveAbsZ(Axis := axZ, Execute := mcMoveAbsZ.Execute, Position := mcMoveAbsZ.Position, Velocity := mcMoveAbsZ.Velocity);

END_FUNCTION_BLOCK

// ---- POUs/FB_IOT.TcPOU
FUNCTION_BLOCK FB_IOT
VAR_INPUT
    iUSS1 : UINT;
    iUSS2 : UINT;
    iUSS3 : UINT;
END_VAR
VAR
    fbMqttClient           : FB_IotMqttClient;
    sMessageToPublish      : STRING(255);
    tmrSendMessageInterval : TON := (PT := T#10S);
    first_cycle            : BOOL := TRUE;
    bStaticPublished       : BOOL := FALSE;
END_VAR

IF first_cycle THEN
    fbMqttClient.sHostName     := '158.180.44.197';
    fbMqttClient.nHostPort     := 1883;
    fbMqttClient.sTopicPrefix  := 'aut/SoSe26/I_bin_da_JJAANN/';
    fbMqttClient.sClientId     := 'I_bin_da_JJAANN-LF';
    fbMqttClient.sUserName     := 'bobm';
    fbMqttClient.sUserPassword := 'letmein';
    first_cycle := FALSE;
END_IF

fbMqttClient.Execute(bConnect := TRUE);

IF fbMqttClient.bConnected THEN
    IF NOT bStaticPublished THEN
        sMessageToPublish := 'I_bin_da_JJAANN';
        fbMqttClient.Publish(sTopic := '$$groupsname', pPayload := ADR(sMessageToPublish), nPayloadSize := LEN(sMessageToPublish) + 1, eQoS := TcIotMqttQos.AtMostOnceDelivery, bRetain := TRUE, bQueue := TRUE);
        sMessageToPublish := 'Doerr Vogel Mueller';
        fbMqttClient.Publish(sTopic := 'names', pPayload := ADR(sMessageToPublish), nPayloadSize := LEN(sMessageToPublish) + 1, eQoS := TcIotMqttQos.AtMostOnceDelivery, bRetain := TRUE, bQueue := TRUE);
        sMessageToPublish := 'g';
        fbMqttClient.Publish(sTopic := 'Fuellstand_rot/$$unit', pPayload := ADR(sMessageToPublish), nPayloadSize := LEN(sMessageToPublish) + 1, eQoS := TcIotMqttQos.AtMostOnceDelivery, bRetain := TRUE, bQueue := TRUE);
        fbMqttClient.Publish(sTopic := 'Fuellstand_blau/$$unit', pPayload := ADR(sMessageToPublish), nPayloadSize := LEN(sMessageToPublish) + 1, eQoS := TcIotMqttQos.AtMostOnceDelivery, bRetain := TRUE, bQueue := TRUE);
        fbMqttClient.Publish(sTopic := 'Fuellstand_gruen/$$unit', pPayload := ADR(sMessageToPublish), nPayloadSize := LEN(sMessageToPublish) + 1, eQoS := TcIotMqttQos.AtMostOnceDelivery, bRetain := TRUE, bQueue := TRUE);
        bStaticPublished := TRUE;
    END_IF

    tmrSendMessageInterval(IN := TRUE);
    IF tmrSendMessageInterval.Q THEN
        tmrSendMessageInterval(IN := FALSE);
        sMessageToPublish := UINT_TO_STRING(iUSS1);
        fbMqttClient.Publish(sTopic := 'Fuellstand_rot', pPayload := ADR(sMessageToPublish), nPayloadSize := LEN(sMessageToPublish) + 1, eQoS := TcIotMqttQos.AtMostOnceDelivery, bRetain := TRUE, bQueue := FALSE);
        sMessageToPublish := UINT_TO_STRING(iUSS2);
        fbMqttClient.Publish(sTopic := 'Fuellstand_blau', pPayload := ADR(sMessageToPublish), nPayloadSize := LEN(sMessageToPublish) + 1, eQoS := TcIotMqttQos.AtMostOnceDelivery, bRetain := TRUE, bQueue := FALSE);
        sMessageToPublish := UINT_TO_STRING(iUSS3);
        fbMqttClient.Publish(sTopic := 'Fuellstand_gruen', pPayload := ADR(sMessageToPublish), nPayloadSize := LEN(sMessageToPublish) + 1, eQoS := TcIotMqttQos.AtMostOnceDelivery, bRetain := TRUE, bQueue := FALSE);
    END_IF
END_IF

END_FUNCTION_BLOCK
